SUBAPPLICATION Uebung_072d_AUI (* GBSD auf UT ausgeben mit AR_Timeout_Zero (Adapter Version) *)
  (* Standard: 61499-2; Description: Copyright (c) 2026 Meisterschulen am Ostbahnhof This program and the accompanying materials are made available under the terms of the Eclipse Public License 2.0 which is available at https://www.eclipse.org/legal/epl-2.0/ SPDX-License-Identifier: EPL-2.0 *)
  (* Version 1.0, 2026-09-17, Franz Höpfinger, Meisterschulen am Ostbahnhof, GBSD mit PHYS Skalierung und AR_Timeout_Zero Fendt-Schaltung (Adapter Version, analog Krauternter TECU_GBSD.SUB) *)
  PACKAGE Uebungen;
  IMPORT Uebungen::const::UT::TECU::DefaultPool_TECU_Numeric::NumberVariable_Ground_based_machine_speed_N;
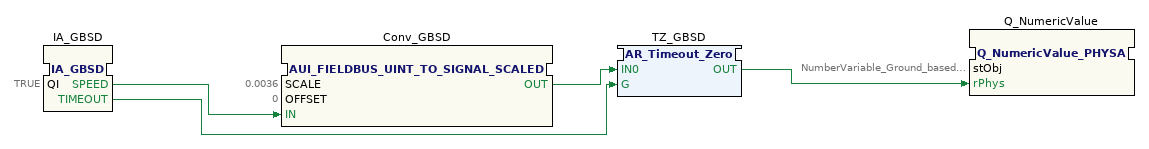
  FBS
    IA_GBSD : isobus::tecu::IA_GBSD(QI := TRUE);
    Conv_GBSD : logiBUS::signalprocessing::fieldbus::AUI_FIELDBUS_UINT_TO_SIGNAL_SCALED(SCALE := 0.0036, OFFSET := 0);
    Q_NumericValue : isobus::UT::Q::Q_NumericValue_PHYSA(stObj := NumberVariable_Ground_based_machine_speed_N);
  END_FBS
  SUBAPPS
    TZ_GBSD : MyLib::sys::AR_Timeout_Zero;
  END_SUBAPPS
  ADAPTER_CONNECTIONS
    IA_GBSD.SPEED TO Conv_GBSD.IN;
    Conv_GBSD.OUT TO TZ_GBSD.IN0;
    IA_GBSD.TIMEOUT TO TZ_GBSD.G;
    TZ_GBSD.OUT TO Q_NumericValue.rPhys;
  END_CONNECTIONS
END_SUBAPPLICATION
